// TIA Portal project "whackamole" (V16)

(* hardware
DEVICE "S7-1200 station_1"  S7-1200 Station
   slot 0: "Rack_0"  S7-1200 Rack  Rack  V1.0
   slot 1: "PLC_1"  CPU 1214C DC/DC/DC  6ES7 214-1AE30-0XB0  V2.2
   slot 3: "AQ 1x12BIT_1"  AQ1 signal board  6ES7 232-4HA30-0XB0  V1.0
*)

// ===== PLC "PLC_1"  CPU 1214C DC/DC/DC =====

VAR_GLOBAL   // PLC tag table "Default tag table"
   "mmm" AT %M0.0 : Bool;
   "oops" AT %M0.1 : Bool;
   "startButton" AT %M0.2 : Bool;
   "Start" AT %M0.3 : Bool;
   "molePop" AT %M0.4 : Bool;
   "newGame" AT %M0.5 : Bool;
   "button1" AT %M0.6 : Bool;
   "button2" AT %M0.7 : Bool;
   "button3" AT %M1.0 : Bool;
   "button4" AT %M1.1 : Bool;
   "lightUp1" AT %M1.2 : Bool;
   "lightUp2" AT %M1.3 : Bool;
   "lightUp3" AT %M1.4 : Bool;
   "lightUp4" AT %M1.5 : Bool;
   "timer1End" AT %M1.6 : Bool;
   "button1Hit" AT %M1.7 : Bool;
   "button2Hit" AT %M2.0 : Bool;
   "button3Hit" AT %M2.1 : Bool;
   "button4Hit" AT %M2.2 : Bool;
   "lightUpHappened" AT %M2.3 : Bool;
   "burh" AT %M2.4 : Bool;
   "clearLight" AT %M2.5 : Bool;
   "newGameButton" AT %M2.6 : Bool;
   "resetArray" AT %M2.7 : Bool;
   "resetTimerArray" AT %M3.0 : Bool;
   "test" AT %M3.1 : Bool;
   "endGame" AT %M3.2 : Bool;
   "resetListCount" AT %M3.3 : Bool;
   "lastValue" AT %MW4 : Int;
   "buttonFlash" AT %M3.4 : Bool;
   "finishFlash" AT %M3.5 : Bool;
   "flash" AT %M3.6 : Bool;
   "flashSecond" AT %M3.7 : Bool;
   "but2" AT %M6.0 : Bool;
   "but1" AT %M6.1 : Bool;
   "but3" AT %M6.2 : Bool;
   "but4" AT %M6.3 : Bool;
   "noFlash" AT %M6.4 : Bool;
END_VAR

DATA_BLOCK "dataList1"   // DB7
{ S7_Optimized_Access := 'TRUE' }
VERSION : 0.1
   VAR
      dataList1 : Array[0..5] of DInt;
   END_VAR
   VAR RETAIN
      buttonList1 : Array[0..3] of DInt;
   END_VAR
BEGIN
   dataList1[0] := 5000;
   dataList1[1] := 10000;
   dataList1[2] := 7000;
   dataList1[3] := 8000;
   dataList1[4] := 12000;
   dataList1[5] := 9000;
   buttonList1[0] := 1;
   buttonList1[1] := 2;
   buttonList1[2] := 3;
   buttonList1[3] := 4;
END_DATA_BLOCK

DATA_BLOCK "dataList2"   // DB8
{ S7_Optimized_Access := 'TRUE' }
VERSION : 0.1
   VAR
      dataList2 : Array[0..5] of DInt;
      buttonList2 : Array[0..3] of DInt;
   END_VAR
BEGIN
   dataList2[0] := 6000;
   dataList2[1] := 9000;
   dataList2[2] := 10000;
   dataList2[3] := 2000;
   dataList2[4] := 8000;
   dataList2[5] := 7000;
   buttonList2[0] := 2;
   buttonList2[1] := 3;
   buttonList2[2] := 1;
   buttonList2[3] := 4;
END_DATA_BLOCK

DATA_BLOCK "dataList3"   // DB9
{ S7_Optimized_Access := 'TRUE' }
VERSION : 0.1
   VAR
      dataList3 : Array[0..5] of DInt;
      buttonList3 : Array[0..3] of DInt;
   END_VAR
BEGIN
   dataList3[0] := 12000;
   dataList3[1] := 8000;
   dataList3[2] := 7000;
   dataList3[3] := 6000;
   dataList3[4] := 7000;
   dataList3[5] := 4000;
   buttonList3[0] := 4;
   buttonList3[1] := 1;
   buttonList3[2] := 3;
   buttonList3[3] := 2;
END_DATA_BLOCK

DATA_BLOCK "currentList"   // DB11
{ S7_Optimized_Access := 'TRUE' }
VERSION : 0.1
   VAR RETAIN
      dataList : Array[0..5] of DInt;
      buttonList : Array[0..3] of DInt;
   END_VAR
BEGIN
END_DATA_BLOCK

// folder: System blocks/Program resources

DATA_BLOCK "numberOfMoles"   // DB1
{ S7_Optimized_Access := 'TRUE' }
AUTHOR : Simatic
FAMILY : IEC
NAME : CNTR
VERSION : 1.0
// stored: InstanceOfName IEC_COUNTER
"IEC_COUNTER"
BEGIN
END_DATA_BLOCK

DATA_BLOCK "timer1"   // DB2
{ S7_Optimized_Access := 'TRUE' }
AUTHOR : Simatic
FAMILY : IEC
NAME : IEC_TMR
VERSION : 1.0
// stored: InstanceOfName IEC_TIMER
"IEC_TIMER"
BEGIN
END_DATA_BLOCK

DATA_BLOCK "timer2"   // DB3
{ S7_Optimized_Access := 'TRUE' }
AUTHOR : Simatic
FAMILY : IEC
NAME : IEC_TMR
VERSION : 1.0
// stored: InstanceOfName IEC_TIMER
"IEC_TIMER"
BEGIN
END_DATA_BLOCK

DATA_BLOCK "timer3"   // DB4
{ S7_Optimized_Access := 'TRUE' }
AUTHOR : Simatic
FAMILY : IEC
NAME : IEC_TMR
VERSION : 1.0
// stored: InstanceOfName IEC_TIMER
"IEC_TIMER"
BEGIN
END_DATA_BLOCK

DATA_BLOCK "timer4"   // DB5
{ S7_Optimized_Access := 'TRUE' }
AUTHOR : Simatic
FAMILY : IEC
NAME : IEC_TMR
VERSION : 1.0
// stored: InstanceOfName IEC_TIMER
"IEC_TIMER"
BEGIN
END_DATA_BLOCK

DATA_BLOCK "totalMoles"   // DB6
{ S7_Optimized_Access := 'TRUE' }
AUTHOR : Simatic
FAMILY : IEC
NAME : CNTR
VERSION : 1.0
// stored: InstanceOfName IEC_COUNTER
"IEC_COUNTER"
BEGIN
END_DATA_BLOCK

DATA_BLOCK "arrayIndex"   // DB10
{ S7_Optimized_Access := 'TRUE' }
AUTHOR : Simatic
FAMILY : IEC
NAME : CNTR
VERSION : 1.0
// stored: InstanceOfName IEC_COUNTER
"IEC_COUNTER"
BEGIN
END_DATA_BLOCK

DATA_BLOCK "listCount"   // DB12
{ S7_Optimized_Access := 'TRUE' }
AUTHOR : Simatic
FAMILY : IEC
NAME : CNTR
VERSION : 1.0
// stored: InstanceOfName IEC_COUNTER
"IEC_COUNTER"
BEGIN
END_DATA_BLOCK

DATA_BLOCK "timerIndex"   // DB13
{ S7_Optimized_Access := 'TRUE' }
AUTHOR : Simatic
FAMILY : IEC
NAME : CNTR
VERSION : 1.0
// stored: InstanceOfName IEC_COUNTER
"IEC_COUNTER"
BEGIN
END_DATA_BLOCK

DATA_BLOCK "lastValueCounter"   // DB14
{ S7_Optimized_Access := 'TRUE' }
AUTHOR : Simatic
FAMILY : IEC
NAME : CNTR
VERSION : 1.0
// stored: InstanceOfName IEC_COUNTER
"IEC_COUNTER"
BEGIN
END_DATA_BLOCK

DATA_BLOCK "flash1"   // DB15
{ S7_Optimized_Access := 'TRUE' }
AUTHOR : Simatic
FAMILY : IEC
NAME : IEC_TMR
VERSION : 1.0
// stored: InstanceOfName IEC_TIMER
"IEC_TIMER"
BEGIN
END_DATA_BLOCK

DATA_BLOCK "flash2"   // DB16
{ S7_Optimized_Access := 'TRUE' }
AUTHOR : Simatic
FAMILY : IEC
NAME : IEC_TMR
VERSION : 1.0
// stored: InstanceOfName IEC_TIMER
"IEC_TIMER"
BEGIN
END_DATA_BLOCK

DATA_BLOCK "flash3"   // DB17
{ S7_Optimized_Access := 'TRUE' }
AUTHOR : Simatic
FAMILY : IEC
NAME : IEC_TMR
VERSION : 1.0
// stored: InstanceOfName IEC_TIMER
"IEC_TIMER"
BEGIN
END_DATA_BLOCK

DATA_BLOCK "flash4"   // DB18
{ S7_Optimized_Access := 'TRUE' }
AUTHOR : Simatic
FAMILY : IEC
NAME : IEC_TMR
VERSION : 1.0
// stored: InstanceOfName IEC_TIMER
"IEC_TIMER"
BEGIN
END_DATA_BLOCK

// folder: (top level)

ORGANIZATION_BLOCK "Main"   // OB1, LAD, ProgramCycle
TITLE = "Main Program Sweep (Cycle)"
{ S7_Optimized_Access := 'TRUE' }
VERSION : 0.1
   VAR_TEMP
      junk : Bool;
   END_VAR
   VAR_TEMP   // added for the SCL form of the ladder/FBD networks
      _w1 : Bool;
   END_VAR
BEGIN

REGION Network 1
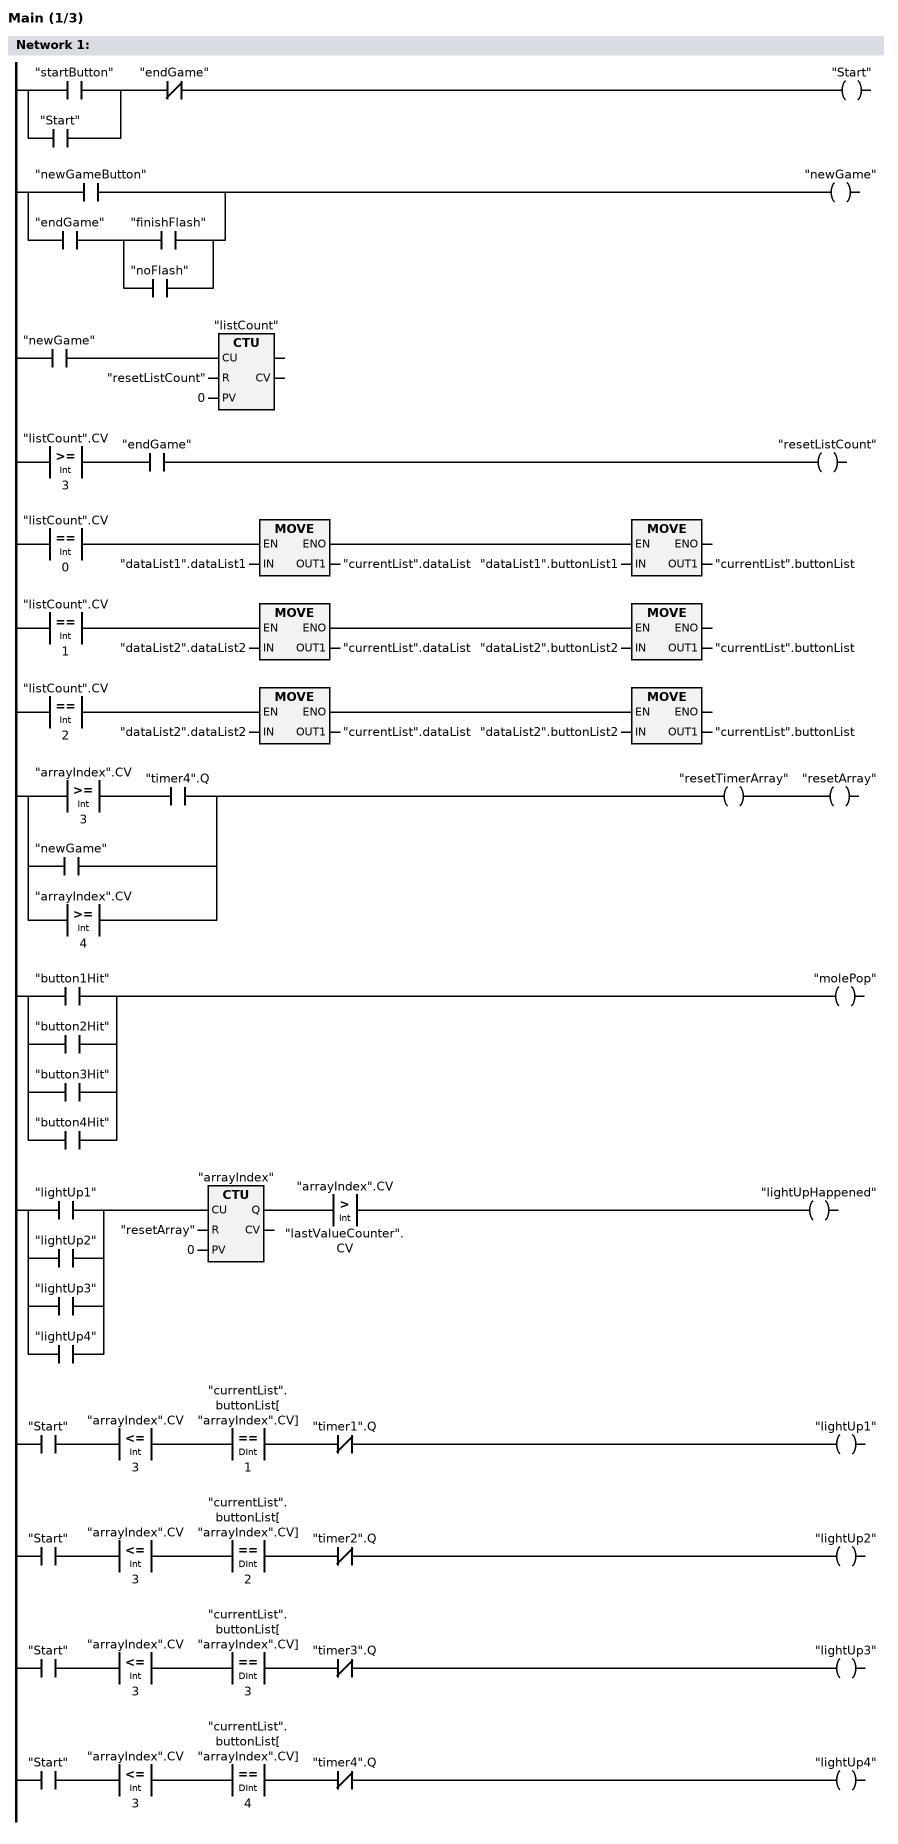
   // ENO of a box is taken as its EN; it also drops when the box reports an error
   "Start" := ("startButton" OR "Start") AND NOT "endGame";
   "newGame" := "newGameButton" OR ("endGame" AND ("finishFlash" OR "noFlash"));
   "listCount".CTU(CU := "newGame", R := "resetListCount", PV := 0);
   "resetListCount" := ("listCount".CV >= 3) AND "endGame";
   IF "listCount".CV = 0 THEN
       "currentList".dataList := "dataList1".dataList1;
       "currentList".buttonList := "dataList1".buttonList1;
   END_IF;
   IF "listCount".CV = 1 THEN
       "currentList".dataList := "dataList2".dataList2;
       "currentList".buttonList := "dataList2".buttonList2;
   END_IF;
   IF "listCount".CV = 2 THEN
       "currentList".dataList := "dataList2".dataList2;
       "currentList".buttonList := "dataList2".buttonList2;
   END_IF;
   "resetTimerArray" := (("arrayIndex".CV >= 3) AND "timer4".Q) OR "newGame" OR ("arrayIndex".CV >= 4);
   "resetArray" := "resetTimerArray";
   "molePop" := "button1Hit" OR "button2Hit" OR "button3Hit" OR "button4Hit";
   "arrayIndex".CTU(CU := "lightUp1" OR "lightUp2" OR "lightUp3" OR "lightUp4", R := "resetArray", PV := 0);
   "lightUpHappened" := "arrayIndex".Q AND ("arrayIndex".CV > "lastValueCounter".CV);
   "lightUp1" := "Start" AND ("arrayIndex".CV <= 3) AND ("currentList".buttonList["arrayIndex".CV] = 1) AND NOT "timer1".Q;
   "lightUp2" := "Start" AND ("arrayIndex".CV <= 3) AND ("currentList".buttonList["arrayIndex".CV] = 2) AND NOT "timer2".Q;
   "lightUp3" := "Start" AND ("arrayIndex".CV <= 3) AND ("currentList".buttonList["arrayIndex".CV] = 3) AND NOT "timer3".Q;
   "lightUp4" := "Start" AND ("arrayIndex".CV <= 3) AND ("currentList".buttonList["arrayIndex".CV] = 4) AND NOT "timer4".Q;
END_REGION

REGION Network 2
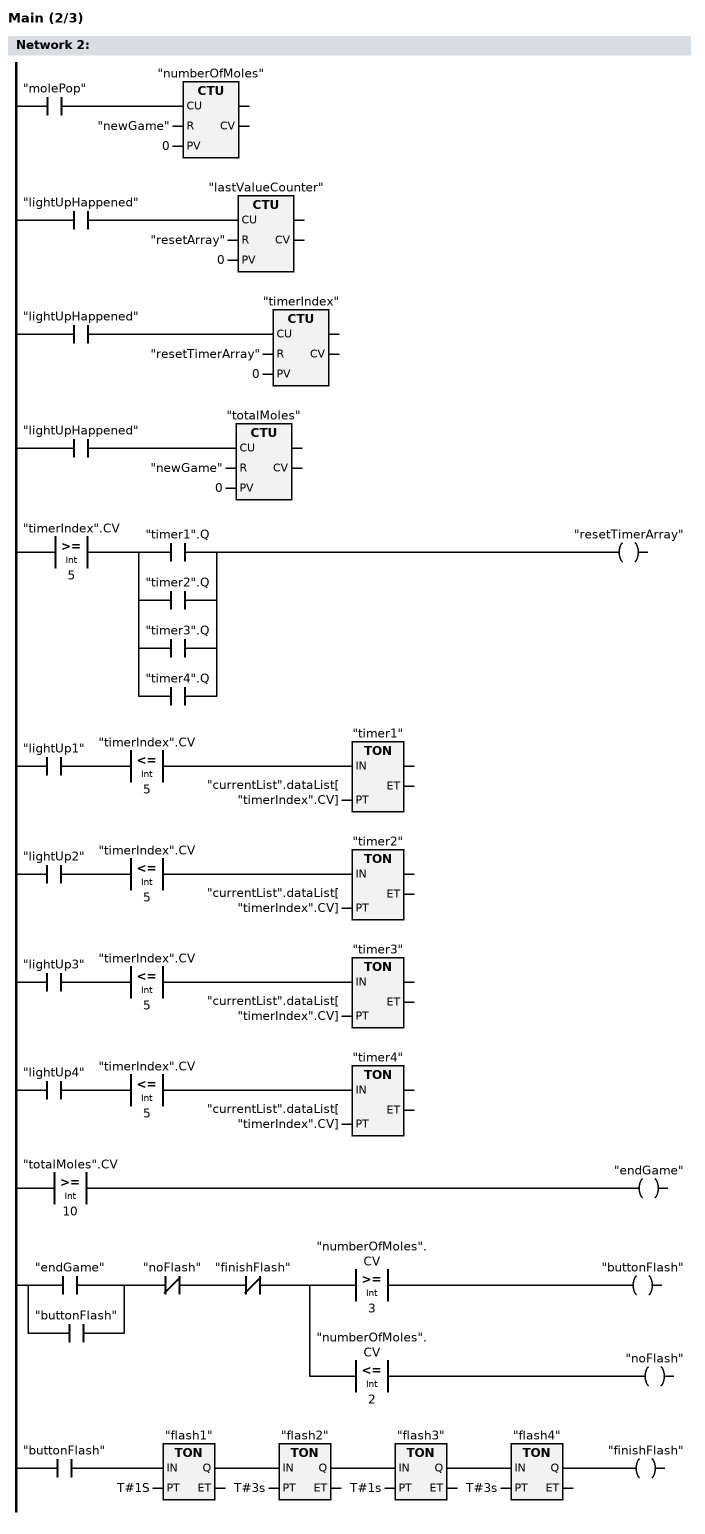
   "numberOfMoles".CTU(CU := "molePop", R := "newGame", PV := 0);
   "lastValueCounter".CTU(CU := "lightUpHappened", R := "resetArray", PV := 0);
   "timerIndex".CTU(CU := "lightUpHappened", R := "resetTimerArray", PV := 0);
   "totalMoles".CTU(CU := "lightUpHappened", R := "newGame", PV := 0);
   "resetTimerArray" := ("timerIndex".CV >= 5) AND ("timer1".Q OR "timer2".Q OR "timer3".Q OR "timer4".Q);
   "timer1".TON(IN := "lightUp1" AND ("timerIndex".CV <= 5), PT := "currentList".dataList["timerIndex".CV]);
   "timer2".TON(IN := "lightUp2" AND ("timerIndex".CV <= 5), PT := "currentList".dataList["timerIndex".CV]);
   "timer3".TON(IN := "lightUp3" AND ("timerIndex".CV <= 5), PT := "currentList".dataList["timerIndex".CV]);
   "timer4".TON(IN := "lightUp4" AND ("timerIndex".CV <= 5), PT := "currentList".dataList["timerIndex".CV]);
   "endGame" := "totalMoles".CV >= 10;
   #_w1 := ("endGame" OR "buttonFlash") AND NOT "noFlash" AND NOT "finishFlash";
   "buttonFlash" := #_w1 AND ("numberOfMoles".CV >= 3);
   "noFlash" := #_w1 AND ("numberOfMoles".CV <= 2);
   "flash1".TON(IN := "buttonFlash", PT := T#1S);
   "flash2".TON(IN := "flash1".Q, PT := T#3s);
   "flash3".TON(IN := "flash2".Q, PT := T#1s);
   "flash4".TON(IN := "flash3".Q, PT := T#3s);
   "finishFlash" := "flash4".Q;
END_REGION

REGION Network 3
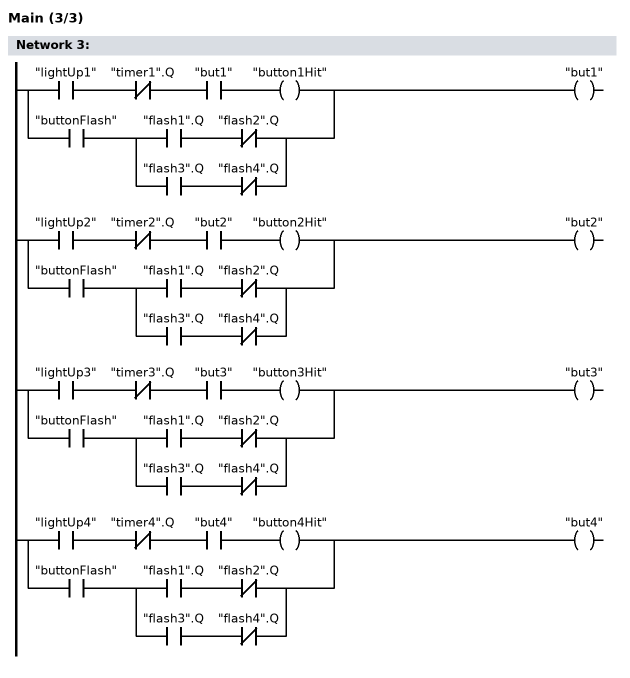
   RUNG wire#powerrail
      Contact( "lightUp1" )
      I_Contact( "timer1".Q )
      Contact( "but1" )
      Coil( "button1Hit" )
      wire#w1
      Coil( "but1" )
   END_RUNG
   RUNG wire#powerrail
      Contact( "buttonFlash" )
      wire#w2
      Contact( "flash1".Q )
      I_Contact( "flash2".Q )
   END_RUNG wire#w1
   RUNG wire#w2
      Contact( "flash3".Q )
      I_Contact( "flash4".Q )
   END_RUNG wire#w1
   RUNG wire#powerrail
      Contact( "lightUp2" )
      I_Contact( "timer2".Q )
      Contact( "but2" )
      Coil( "button2Hit" )
      wire#w3
      Coil( "but2" )
   END_RUNG
   RUNG wire#powerrail
      Contact( "buttonFlash" )
      wire#w4
      Contact( "flash1".Q )
      I_Contact( "flash2".Q )
   END_RUNG wire#w3
   RUNG wire#w4
      Contact( "flash3".Q )
      I_Contact( "flash4".Q )
   END_RUNG wire#w3
   RUNG wire#powerrail
      Contact( "lightUp3" )
      I_Contact( "timer3".Q )
      Contact( "but3" )
      Coil( "button3Hit" )
      wire#w5
      Coil( "but3" )
   END_RUNG
   RUNG wire#powerrail
      Contact( "buttonFlash" )
      wire#w6
      Contact( "flash1".Q )
      I_Contact( "flash2".Q )
   END_RUNG wire#w5
   RUNG wire#w6
      Contact( "flash3".Q )
      I_Contact( "flash4".Q )
   END_RUNG wire#w5
   RUNG wire#powerrail
      Contact( "lightUp4" )
      I_Contact( "timer4".Q )
      Contact( "but4" )
      Coil( "button4Hit" )
      wire#w7
      Coil( "but4" )
   END_RUNG
   RUNG wire#powerrail
      Contact( "buttonFlash" )
      wire#w8
      Contact( "flash1".Q )
      I_Contact( "flash2".Q )
   END_RUNG wire#w7
   RUNG wire#w8
      Contact( "flash3".Q )
      I_Contact( "flash4".Q )
   END_RUNG wire#w7
   // the same network as SCL:
   "button1Hit" := "lightUp1" AND NOT "timer1".Q AND "but1";
   "but1" := "button1Hit" OR ("buttonFlash" AND (("flash1".Q AND NOT "flash2".Q) OR ("flash3".Q AND NOT "flash4".Q)));
   "button2Hit" := "lightUp2" AND NOT "timer2".Q AND "but2";
   "but2" := "button2Hit" OR ("buttonFlash" AND (("flash1".Q AND NOT "flash2".Q) OR ("flash3".Q AND NOT "flash4".Q)));
   "button3Hit" := "lightUp3" AND NOT "timer3".Q AND "but3";
   "but3" := "button3Hit" OR ("buttonFlash" AND (("flash1".Q AND NOT "flash2".Q) OR ("flash3".Q AND NOT "flash4".Q)));
   "button4Hit" := "lightUp4" AND NOT "timer4".Q AND "but4";
   "but4" := "button4Hit" OR ("buttonFlash" AND (("flash1".Q AND NOT "flash2".Q) OR ("flash3".Q AND NOT "flash4".Q)));
END_REGION
END_ORGANIZATION_BLOCK